FUNCTION_BLOCK ConveyorCTLMultiCast (* Basic Function Block Type *)
  (* Standard: 61499-2 *)
  (* Version 0.2, 2003-12-04, JHC, Rockwell Automation, Renamed for better indexing. *)
  (* Version 0.1, 2002-11-05, JHC, Rockwell Automation, Corrected missing ST element in Algorithm REQ. *)
  (* Version 0.0, 2000-05-30, JHC, Rockwell Automation *)
  (* Compiler header: package fb.rt.cs725; *)
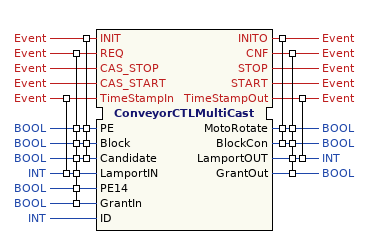
  EVENT_INPUT
    INIT WITH PE, Block, Candidate; (* Initialization Request *)
    REQ WITH PE, Block, Candidate, GrantIn, LamportIN, PE14; (* Normal Execution Request *)
    CAS_STOP;
    CAS_START;
    TimeStampIn WITH LamportIN;
  END_EVENT
  EVENT_OUTPUT
    INITO WITH MotoRotate, BlockCon; (* Initialization Confirm *)
    CNF WITH MotoRotate, BlockCon, LamportOUT, GrantOut; (* Execution Confirmation *)
    STOP;
    START;
    TimeStampOut WITH LamportOUT;
  END_EVENT
  VAR_INPUT
    PE : BOOL; (* Input event qualifier *)
    Block : BOOL;
    Candidate : BOOL;
    LamportIN : INT;
    PE14 : BOOL;
    GrantIn : BOOL;
    ID : INT;
  END_VAR
  VAR_OUTPUT
    MotoRotate : BOOL; (* Output event qualifier *)
    BlockCon : BOOL;
    LamportOUT : INT;
    GrantOut : BOOL;
  END_VAR
  VAR
    lastPE : BOOL := 1;
    lastBlock : BOOL := 0;
    lamportClock : INT;
    delayStop : INT;
  END_VAR
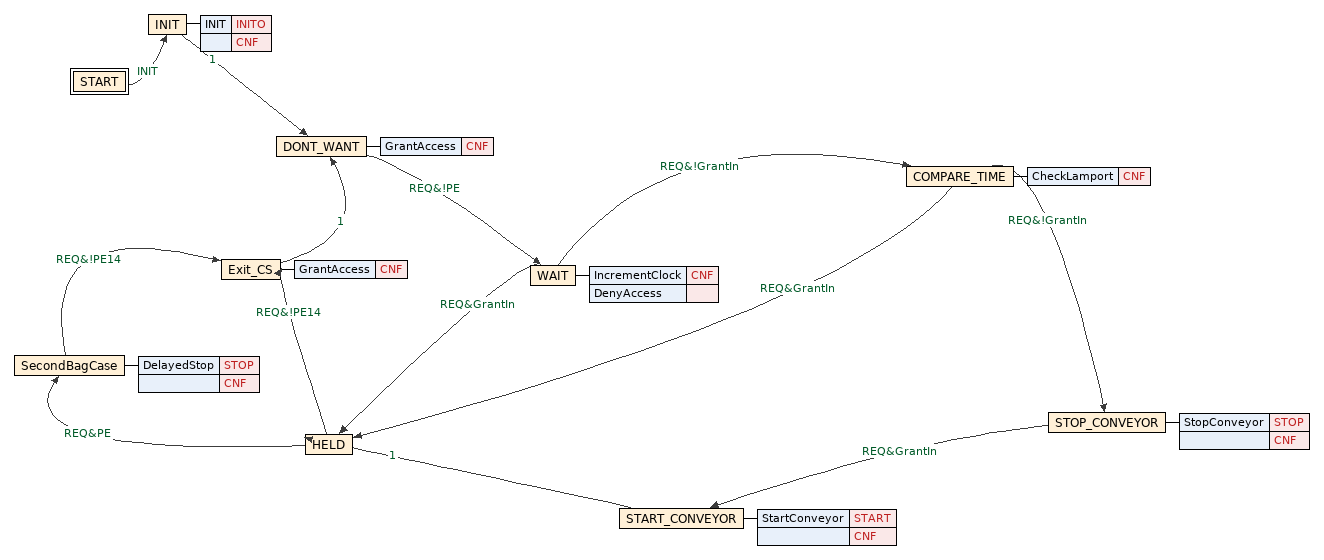
  EC_STATES
    START; (* Initial State *)
    INIT : INIT -> INITO, -> CNF; (* Initialization *)
    DONT_WANT : GrantAccess -> CNF;
    WAIT : IncrementClock -> CNF, DenyAccess;
    HELD; (* Inside Critical Section *)
    Exit_CS : GrantAccess -> CNF;
    COMPARE_TIME : CheckLamport -> CNF;
    STOP_CONVEYOR : StopConveyor -> STOP, -> CNF;
    START_CONVEYOR : StartConveyor -> START, -> CNF;
    SecondBagCase : DelayedStop -> STOP, -> CNF;
  END_STATES
  EC_TRANSITIONS
    START TO INIT := INIT;
    INIT TO DONT_WANT := 1;
    DONT_WANT TO WAIT := REQ&!PE;
    WAIT TO HELD := REQ&GrantIn;
    HELD TO Exit_CS := REQ&!PE14;
    Exit_CS TO DONT_WANT := 1;
    WAIT TO COMPARE_TIME := REQ&!GrantIn;
    COMPARE_TIME TO STOP_CONVEYOR := REQ&!GrantIn;
    COMPARE_TIME TO HELD := REQ&GrantIn;
    STOP_CONVEYOR TO START_CONVEYOR := REQ&GrantIn;
    START_CONVEYOR TO HELD := 1;
    HELD TO SecondBagCase := REQ&PE;
    SecondBagCase TO Exit_CS := REQ&!PE14;
  END_TRANSITIONS
  ALGORITHM INIT IN ST: (* Initialization algorithm *)
MotoRotate := TRUE;
Block := FALSE;
lamportClock := 0;
GrantOut := FALSE;
delayStop := 0;


System.out.println("Conveyor: "+ID+" Multicast INIT");
  END_ALGORITHM
  ALGORITHM REQ IN ST: (* Normally executed algorithm *)
System.out.println(this +  " -> Candidate" + Candidate);
IF Candidate THEN
IF lastPE !:= PE THEN
IF NOT PE THEN
BlockCon:= TRUE;
System.out.println("BlockCon = true");
ELSE
BlockCon:=FALSE;
System.out.println("BlockCon = false");
END_IF
lastPE := PE;
END_IF
IF lastBlock !:= Block THEN
IF Block THEN
STOP.serviceEvent(this);
MotoRotate := FALSE;
System.out.println("Cas Stop");
ELSE
START.serviceEvent(this);
MotoRotate := TRUE;
System.out.println("Cas Start");
END_IF
lastBlock := Block;
END_IF
END_IF
  END_ALGORITHM
  ALGORITHM START IN ST:
MotoRotate:=TRUE;
System.out.println(this + " Start " + MotoRotate);

System.out.println("Start " + MotoRotate);
  END_ALGORITHM
  ALGORITHM STOP IN ST:
MotoRotate := FALSE;
System.out.println(this + " Stop " + MotoRotate);

System.out.println("Stop " + MotoRotate);
  END_ALGORITHM
  ALGORITHM CheckLamport IN Java:
System.out.println("Conveyor: "+ ID.value +" LamportIN:"+ LamportIN.value + " LAMPORTCLK:" +lamportClock.value);

if(LamportIN.value > lamportClock.value){
GrantOut.value = true;
System.out.println(ID.value + " Own LamportClock is smaller!");
}else{
GrantOut.value = false;
System.out.println(ID.value + " Lamport IN is smaller!");
}
  END_ALGORITHM
  ALGORITHM IncrementClock IN Java:
lamportClock.value++;
LamportOUT.value = lamportClock.value;
  END_ALGORITHM
  ALGORITHM GrantAccess IN Java:
System.out.println("Conveyor: "+ID.value+ " grants access");

GrantOut.value = true;
delayStop.value = 0;
  END_ALGORITHM
  ALGORITHM StopConveyor IN Java:
System.out.println("Conveyor: "+ID.value + " Stop Conveyor Multicast!");
MotoRotate.value = false;
  END_ALGORITHM
  ALGORITHM StartConveyor IN Java:
GrantOut.value = false;

MotoRotate.value = true;
System.out.println("Conveyor: "+ID.value +" Start Conveyer Multicast");
  END_ALGORITHM
  ALGORITHM ResetLamport IN Java:
lamportClock.value = 0;
System.out.println("Conveyor: "+ ID.value + " Reset the Lamport Clock");
  END_ALGORITHM
  ALGORITHM DenyAccess IN Java:
GrantOut.value = false;
  END_ALGORITHM
  ALGORITHM DelayedStop IN Java:
if(delayStop.value >= 10){
System.out.println("Conveyor: "+ID.value + " Stop Conveyor Multicast!");
MotoRotate.value = false;
}else{
delayStop.value++;
}
  END_ALGORITHM
END_FUNCTION_BLOCK
